Staubli VAL3: OnF7.pgx

program OnF7()
begin
  //

end
